// Mitsubishi GX Works2 project: Bobinadora   PLC: FX1N/FX1NC

PROGRAM MAIN
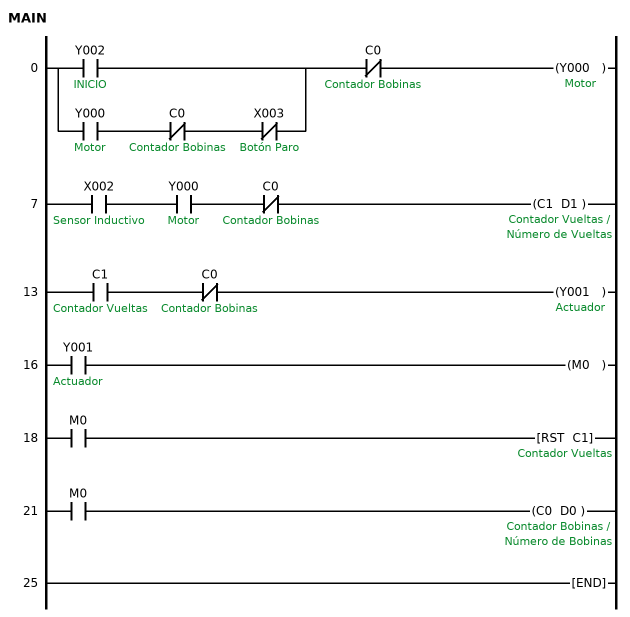
0     LD      Y002  ; INICIO
      LD      Y000  ; Motor
      ANI     C0  ; Contador Bobinas
      ANI     X003  ; Botón Paro
      ORB
      ANI     C0  ; Contador Bobinas
      OUT     Y000  ; Motor
7     LD      X002  ; Sensor Inductivo
      AND     Y000  ; Motor
      ANI     C0  ; Contador Bobinas
      OUT     C1 D1  ; Contador Vueltas / Número de Vueltas
13    LD      C1  ; Contador Vueltas
      ANI     C0  ; Contador Bobinas
      OUT     Y001  ; Actuador
16    LD      Y001  ; Actuador
      OUT     M0
18    LD      M0
      RST     C1  ; Contador Vueltas
21    LD      M0
      OUT     C0 D0  ; Contador Bobinas / Número de Bobinas
25    END
END_PROGRAM

// device comments not shown above
X000  ; Botón Inicio Principal
X001  ; Botón Inicio Bobinas
